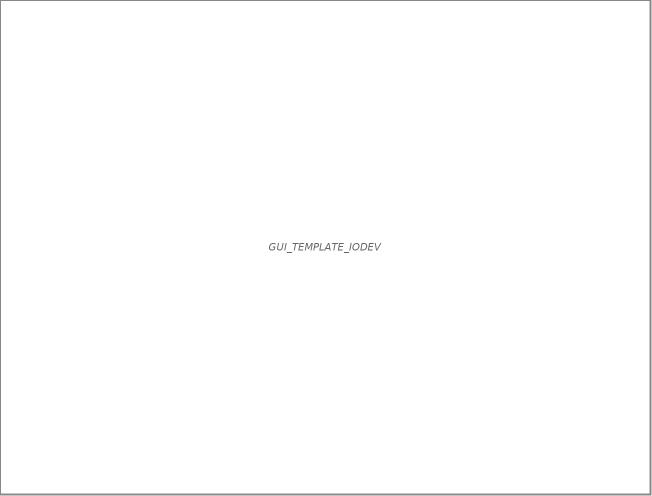
VISUALIZATION GUI_IODev001  // 652x496
    Frame (0,0 650x494)
        shows GUI_TEMPLATE_IODEV(m_Instance := MAIN.IODev001)
END_VISUALIZATION

(* stored: Version 1.1.0.1, ProductVersion 3.1.4024.3
   Visu GUI_IODev001: Id {ba6b4829-cfe8-4c1b-80a7-d8c3b6d4dc60} *)
